FUNCTION_BLOCK FB_SimulatedOutClose_DG IMPLEMENTS ITF_Regelschuif_OutClose_DG
VAR
	internalState : BOOL := FALSE;
END_VAR

{warning 'Add method implementation '}
METHOD set : BOOL
VAR_INPUT
	state : BOOL;
END_VAR
internalState := state;
END_METHOD

END_FUNCTION_BLOCK

(* stored: Version 1.1.0.1, ProductVersion 3.1.4026.8
   POU FB_SimulatedOutClose_DG: Id {0b2b4ec8-8f4a-4501-a03d-729d4fad0c8c}, SpecialFunc None
   Method set: Id {117eb3f5-f304-4f28-b5f9-9fe807e54b8d} *)
